PROGRAM PRG_LI3K2_K2B
VAR
    {attribute 'pytmc' := 'pv: LI3K2:K2B'}
    fbLI3K2: FB_LIC;

    fbStateSetup: FB_StateSetupHelper;
    stDefault: ST_PositionState := (
        fVelocity := 1,
        bMoveOk := TRUE,
        bValid := TRUE
    );
END_VAR


fbStateSetup(stPositionState:=stDefault, bSetDefault:=TRUE);

fbStateSetup(stPositionState:=fbLI3K2.stOut, fPosition:=0.118, sPmpsState:='LI3K2:K2B-OUT');
fbStateSetup(stPositionState:=fbLI3K2.stMirror1, fPosition:=-36.38, sPmpsState:='LI3K2:K2B-MIRROR1');
fbStateSetup(stPositionState:=fbLI3K2.stMirror2, fPosition:=-70.38, sPmpsState:='LI3K2:K2B-MIRROR2');
fbStateSetup(stPositionState:=fbLI3K2.stTarget1, fPosition:=-102.38, sPmpsState:='LI3K2:K2B-TARGET1');

fbLI3K2(
    fbFFHWO := GVL.fbFastFaultOutput2,
    fbArbiter := GVL.fbArbiter2,
    stYStage := Main.M21,
    sDeviceName := 'LI3K2:K2B',
    sTransitionKey := 'LI3K2:K2B-TRANSITION',
    bEnableMotion := TRUE,
    bEnableBeamParams := TRUE,
    bEnablePositionLimits := TRUE,
);

END_PROGRAM

(* stored: Version 1.1.0.1, ProductVersion 3.1.4022.18
   POU PRG_LI3K2_K2B: Id {2a0870d4-376e-46af-943a-d045301a70c9}, SpecialFunc None *)
